(* Logix 5000 project; controller miPrimerPrograma Emulate 5570 rev 32.11; software revision 32.02 *)

TASK T00_MainTask (continuous, watchdog 500 ms) : P00_MainProgram

MODULES
   Local : Emulate 5570 (ICP 2, rev 32.11)
END_MODULES

VAR_GLOBAL   (* controller tags *)
   entrada1 : BOOL;   // memoriaVirtual
   entrada2 : BOOL;   // memoriaVirtual
   salida1 : BOOL;   // memoriaVirual
END_VAR

PROGRAM P00_MainProgram   (* main routine R00_MainRoutine *)

ROUTINE R00_MainRoutine   (* ladder *)
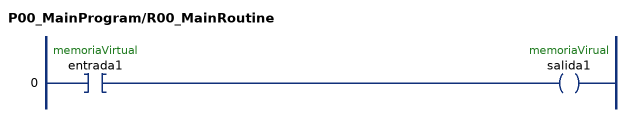
   0: XIC(entrada1)OTE(salida1);
END_ROUTINE
END_PROGRAM
